PROGRAM PRG_Servo1
VAR
	nState: INT;
	bBaslat	: bool;
	bSensor1: BOOL;
	rSayici: R_TRIG;
	bSensor2: BOOL;
	nSayici: INT;
	nCounter: INT;
END_VAR

stAxis1.INPUT.bEnable	:= TRUE;
staxis1.INPUT.bStop:=FALSE;
stAxis1.INPUT.bReset := FALSE;


rSayici(CLK:= bSensor2, Q=> );
CASE nState OF
	
0:
	IF bBaslat AND staxis1.OUTPUT.bEnabled AND NOT stAxis1.OUTPUT.bPowerErr THEN
		nState	:= 10;
		nCounter := 0;
	END_IF
	
10:
	stAxis1.INPUT.bMoveAbs	:= TRUE;
	stAxis1.INPUT.fVelocity	:= 4000;
	stAxis1.INPUT.fPosition	:= 30000;
	
	IF stAxis1.OUTPUT.bMoveAbsBusy AND NOT stAxis1.OUTPUT.bMoveAbsErr THEN

		nState					:= 20;
		stAxis1.INPUT.bMoveAbs:=FALSE;

	ELSIF stAxis1.OUTPUT.bMoveAbsErr THEN
	
	nState					:= 999;
	nCounter := nState;
	stAxis1.INPUT.bMoveAbs	:= FALSE;

	END_IF
			
20:
	IF stAxis1.OUTPUT.bMoveAbsDone AND NOT stAxis1.OUTPUT.bMoveAbsErr THEN
		nState					:= 30;
		nCounter := nState;

	ELSIF stAxis1.OUTPUT.bMoveAbsErr THEN	
		nState					:= 999;
		nCounter := nState;

	END_IF
	
30:	
	IF bSensor1 THEN
		nState	:= 40;
		nCounter:=nState;
	END_IF
	
40:
	nCounter:=30;

	stAxis1.INPUT.bMoveAbs	:= TRUE;
	stAxis1.INPUT.fVelocity	:= 7000;
	stAxis1.INPUT.fPosition	:= 50000;
	
	IF stAxis1.OUTPUT.bMoveAbsBusy AND NOT stAxis1.OUTPUT.bMoveAbsErr THEN
		stAxis1.INPUT.bMoveAbs	:= FALSE;
		nState					:= 50;

	ELSIF stAxis1.OUTPUT.bMoveAbsErr THEN
		nState					:= 999;
		nCounter := nState;

		stAxis1.INPUT.bMoveAbs	:= FALSE;		
	END_IF
	
50:
	IF stAxis1.OUTPUT.bMoveAbsDone AND NOT stAxis1.OUTPUT.bMoveAbsErr THEN
		nState					:= 60;
		nCounter := nState;

	ELSIF stAxis1.OUTPUT.bMoveAbsErr THEN	
		nState					:= 999;
		nCounter := nState;

	END_IF

60:
	IF rSayici.Q AND nSayici<5 THEN
		nSayici	:= nSayici+1;	
	ELSIF nSayici>=5 THEN
		nSayici	:=0;
		nState	:= 70;
		nCounter := nState;
	END_IF

70:
	stAxis1.INPUT.bMoveAbs	:= TRUE;

	stAxis1.INPUT.fVelocity	:= 8000;
	stAxis1.INPUT.fPosition	:= 0;
	nCounter:=60;
	IF stAxis1.OUTPUT.bMoveAbsBusy AND NOT stAxis1.OUTPUT.bMoveAbsErr THEN
		stAxis1.INPUT.bMoveAbs	:= FALSE;
		nState					:= 80;
		nCounter := nState;

	ELSIF stAxis1.OUTPUT.bMoveAbsErr THEN
		nState					:= 999;
		nCounter := nState;

		stAxis1.INPUT.bMoveAbs	:= FALSE;		
	END_IF
	
80:
	IF stAxis1.OUTPUT.bMoveAbsDone AND NOT stAxis1.OUTPUT.bMoveAbsErr THEN
				nState	:= 0;
				nCounter := nState;

	ELSIF stAxis1.OUTPUT.bMoveAbsErr THEN	
		nState					:= 999;
		nCounter := nState;

	END_IF
	
END_CASE

IF stAxis1.OUTPUT.bPowerErr THEN
	stAxis1.INPUT.bReset := TRUE;
	nState:=0;
END_IF

IF NOT bBaslat THEN
	
staxis1.INPUT.bStop:=TRUE;
stAxis1.INPUT.bMoveAbs	:= FALSE;
staxis1.OUTPUT.bEnabled:=TRUE;


		IF staxis1.OUTPUT.bEnabled
		AND NOT stAxis1.OUTPUT.bPowerErr 
		AND NOT stAxis1.OUTPUT.bMoveAbsErr
		AND NOT staxis1.OUTPUT.bStopErr 
		AND  staxis1.OUTPUT.bStopBusy THEN
	
	staxis1.INPUT.bStop:=FALSE;
	nState:=nCounter;

	END_IF

END_IF

END_PROGRAM

(* stored: Version 1.1.0.1, ProductVersion 3.1.4022.18
   POU PRG_Servo1: Id {3613d12f-9e52-4b46-b051-619bcd6c45f5}, SpecialFunc None *)
